FUNCTION "StringToReal" : Void
{ S7_Optimized_Access := 'TRUE' }
VERSION : 0.1
   VAR_INPUT
      In : String;
   END_VAR

   VAR_OUTPUT
      Out : Real;
   END_VAR


BEGIN
	#Out := STRING_TO_REAL(#In);
END_FUNCTION

